// TIA Portal V18 export
DATA_BLOCK "ServoV90_DeviceCtl"   // DB4073
{ S7_Optimized_Access := 'FALSE' }
// stored: AutoNumber false
   VAR RETAIN
      V90Servo : Array[1..4] of Struct
         i : Int;
         nError : Int;
         nWarning : Int;
         nPositionListNo : Int;
         Pos : "PosList";
         Point : Array[0..39] of Struct
            Start : Bool;
            Achieve : Bool;
         END_STRUCT;
      END_STRUCT;
   END_VAR
BEGIN
   V90Servo[1..4].nPositionListNo := 1;
   // V90Servo[1].Pos.List[1] : 待机位
   // V90Servo[1].Pos.List[2] : 排钉位
   // V90Servo[1].Pos.List[3] : 第一个颗螺钉位置
   // V90Servo[1].Pos.List[4] : 第二个颗螺钉位置
   // V90Servo[2].Pos.List[1] : 待机位
   // V90Servo[2].Pos.List[2] : 排钉位
   // V90Servo[2].Pos.List[3] : 第一个颗螺钉位置
   // V90Servo[2].Pos.List[4] : 第二个颗螺钉位置
   V90Servo[1].Pos.List[4..19].Pos := 0;
   V90Servo[1].Pos.List[3..19].Vel := 0;
   // V90Servo[1].Point[1] : 初始位 / 上料位1
   // V90Servo[1].Point[2] : 抓料位 / 上料位2
   // V90Servo[1].Point[3] : 上料拍照位 / 上料位3
   // V90Servo[1].Point[4] : 下料位1 / 上料位4
   // V90Servo[1].Point[5] : 下料位2 / 上料位5
   // V90Servo[1].Point[6] : 下料位3 / 上料位6
   // V90Servo[1].Point[7] : 下料位4 / 上料位7
   // V90Servo[1].Point[8] : 下料位5 / 上料位8
   // V90Servo[1].Point[9] : NG下料位
   // V90Servo[2].Point[1] : 初始位
   // V90Servo[2].Point[2] : 取料位1 / 扫码位置2
   // V90Servo[2].Point[3] : 取料位2 / 扫码位置3
   // V90Servo[2].Point[4] : 取料位3 / 扫码位置4
   // V90Servo[2].Point[5] : 取料位4 / 扫码位置5
   // V90Servo[2].Point[6] : 取料位5 / 扫码位置6
   // V90Servo[2].Point[7] : 清洁位 / 扫码位置7
   // V90Servo[2].Point[8] : NG位 / 扫码位置8
   // V90Servo[2].Point[9] : 快速装配位
   // V90Servo[2].Point[10] : 慢速装配位
END_DATA_BLOCK
